Yaskawa INFORM job: SEND-SHIFT-FRONT-S1.JBI

/JOB
//NAME SEND-SHIFT-FRONT-S1
//POS
///NPOS 0,0,0,1,0,0
///USER 10
///TOOL 1
///POSTYPE USER
///RECTAN
///RCONF 0,0,0,0,0,0,0,0,0,0,0,0,0,0,0,0,0,0,0,0,0,0,0,0
P00173=2.671,-1.737,-1.666,90.0000,0.0004,89.9986
//INST
///DATE 2018/09/04 08:22
///ATTR SC,RW
NOP
'***** send shift value
GETE D067 P0173 (1)
DIV D067 100
MACRO1 MJ#(2) ARGF100 ARGF67
END
